Staubli VAL3: CartesianAccel.pjx

--- CartesianAccel.pjx ---
Parameters version=s7.9.1 stackSize=5000 millimeterUnit=true
Data file=CartesianAccel.dtx

--- CartesianAccel.dtx ---
public num ax
public num ay
public num az
public num arx
public num ary
public num arz
